INTERFACE I_Nasmyth

METHOD SetNasmyth : BOOL
VAR_INPUT
	Port	: INT;
END_VAR
END_METHOD

END_INTERFACE

(* stored: Version 1.1.0.1, ProductVersion 3.1.4024.12
   Itf I_Nasmyth: Id {3d5a95db-dda5-4c5c-90eb-98d64d4dd740}
   Method SetNasmyth: Id {b269bb4f-772b-443e-acef-1282c6633bcc} *)
